
// ===== library: MasterCopy "Flow_Sensor" =====

FUNCTION_BLOCK "Flow_Sensor"   // FB1, FBD
TITLE = Pulsed Output Flow Accumlation
{ S7_Optimized_Access := 'TRUE' }
VERSION : 0.1
// Description: This function is used to Accumlate the flow passing through a pulsed-output flow sensor connected to the digital input channel with the address#Flow_Meter.
// Author: Ahmed Abd Alrahiem
// Email: a.abdalrahiem@gmail.com
// Last Modification Date: July 21, 2021
   VAR_INPUT
      Flow_Meter : Bool;   // The adress of the digital input channel which the Flow sensor is connected to
      pulses_per_litre : UInt;   // The number of pulses which the sesnor will provide after having one letre through it
      Reset : Bool;   // If set, the accumlated flow will be reset to 0
   END_VAR
   VAR_OUTPUT
      Accumlated_Flow : Real;   // The accumlated flow passing through the sensor
   END_VAR
   VAR RETAIN
      pos_edge1 : Bool;
      Flow_FB_counter_DB : CTU_UINT;
   END_VAR
   VAR_TEMP
      OF_DN : Bool;
      counted_pulses : UInt;
      Accumlated_Flow_temp : Real;
      Flow_base : Real;
      Flow_Delta : Real;
   END_VAR
   VAR_TEMP   // added for the SCL form of the ladder/FBD networks
      _w1 : Bool;
   END_VAR
BEGIN

REGION Network 1: Pulse Counting
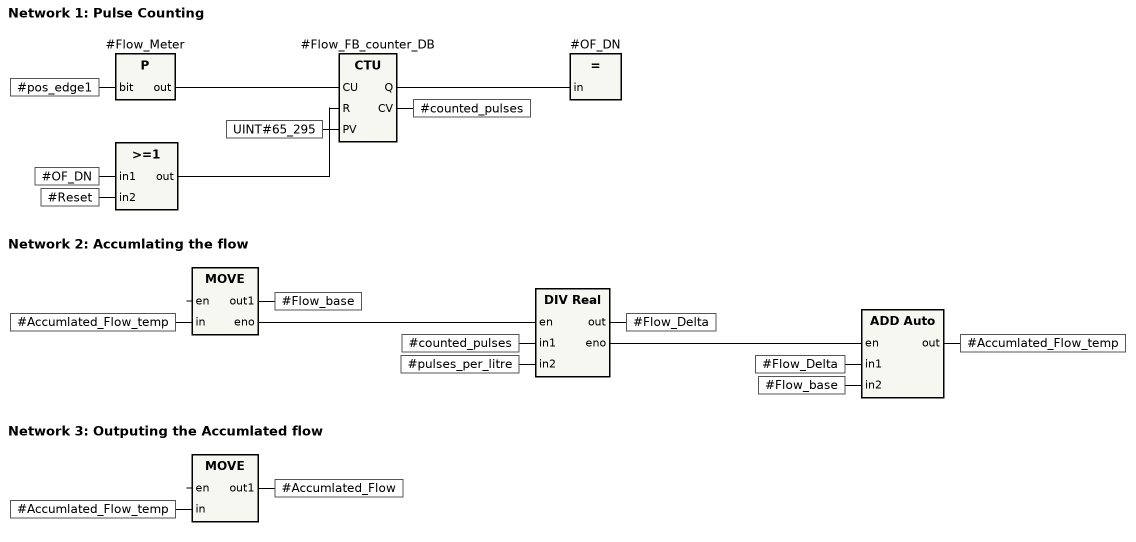
   #_w1 := #Flow_Meter AND NOT #pos_edge1;   // rising edge of #Flow_Meter
   #pos_edge1 := #Flow_Meter;
   #Flow_FB_counter_DB(CU := #_w1, R := #OF_DN OR #Reset, PV := UINT#65_295, CV => #counted_pulses);   // CTU
   #OF_DN := #Flow_FB_counter_DB.Q;
END_REGION

REGION Network 2: Accumlating the flow
   // The flow is accumlated, with integer overflow avoidance
   // ENO of a box is taken as its EN; it also drops when the box reports an error
   #Flow_base := #Accumlated_Flow_temp;
   #Flow_Delta := #counted_pulses / #pulses_per_litre;
   #Accumlated_Flow_temp := #Flow_Delta + #Flow_base;
END_REGION

REGION Network 3: Outputing the Accumlated flow
   #Accumlated_Flow := #Accumlated_Flow_temp;
END_REGION
END_FUNCTION_BLOCK

// ===== library: MasterCopy "Flow_Rate_Sensor" =====

FUNCTION_BLOCK "Flow_Rate_Sensor"   // FB2, FBD
TITLE = Flow rate calculation of a pulsed-output flow sensor
{ S7_Optimized_Access := 'TRUE' }
VERSION : 0.1
// Description: This function is used to calculate the frequecy of the pulses and convert it to the flow rate.
// Author: Ahmed Abd Alrahiem
// Email: a.abdalrahiem@gmail.com
// Last Modification Date: July 21, 2021
   VAR_INPUT
      Flow_Meter : Bool;   // The adress of the digital input channel which the Flow sensor is connected to
      "HZ_per_litre/min" : UInt;   // The proportionality constant between the pulse frequency and the flow rate
      Integration_Time : Time;   // The time window (in sec) used for flow rate calculation, it should be at least higher than the least possible pulse duration
   END_VAR
   VAR_OUTPUT
      Flow_Rate : Real;   // The flow rate of the stream passing through the sensor, calculated over the integration time
   END_VAR
   VAR RETAIN
      pos_edge1 : Bool;
      OF_DN : Bool;
      Flow_FB_counter_DB : CTU_UDINT;
      Flow_Rate_FB_Timer_DB : TP_TIME;
      Always_True : Bool := True;
   END_VAR
   VAR_TEMP
      Int_Time_DN : Bool;
      Integration_Time_Uint : UInt;
      Frequency : Real;
      counted_pulses : UDInt;
      counted_pulses_real : Real;
   END_VAR
   VAR_TEMP   // added for the SCL form of the ladder/FBD networks
      _w1 : Bool;
   END_VAR
BEGIN

REGION Network 1: Pulses counting
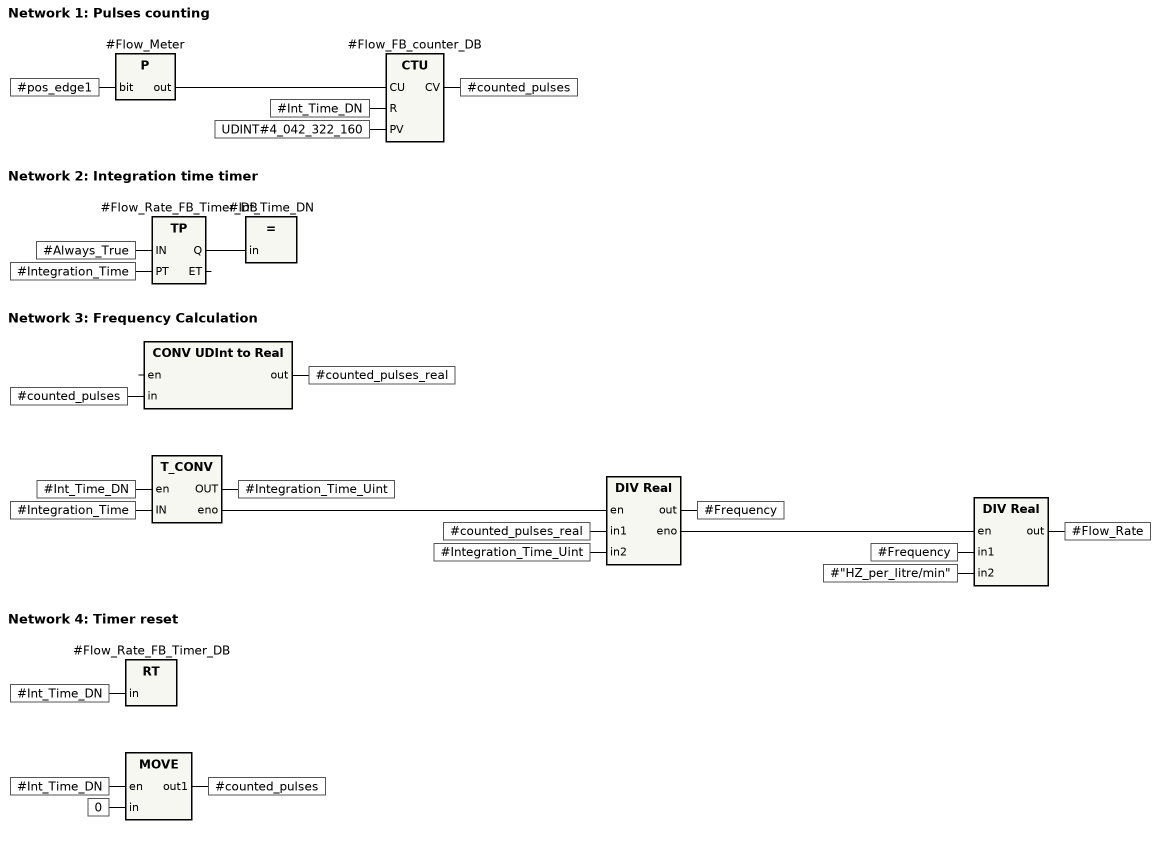
   #_w1 := #Flow_Meter AND NOT #pos_edge1;   // rising edge of #Flow_Meter
   #pos_edge1 := #Flow_Meter;
   #Flow_FB_counter_DB(CU := #_w1, R := #Int_Time_DN, PV := UDINT#4_042_322_160, CV => #counted_pulses);   // CTU
END_REGION

REGION Network 2: Integration time timer
   #Flow_Rate_FB_Timer_DB(IN := #Always_True, PT := #Integration_Time);   // TP
   #Int_Time_DN := #Flow_Rate_FB_Timer_DB.Q;
END_REGION

REGION Network 3: Frequency Calculation
   // ENO of a box is taken as its EN; it also drops when the box reports an error
   #counted_pulses_real := UDINT_TO_REAL(#counted_pulses);
   IF #Int_Time_DN THEN
       #Integration_Time_Uint := T_CONV(IN := #Integration_Time);
       #Frequency := #counted_pulses_real / #Integration_Time_Uint;
       #Flow_Rate := #Frequency / #"HZ_per_litre/min";
   END_IF;
END_REGION

REGION Network 4: Timer reset
   IF #Int_Time_DN THEN
       RESET_TIMER(#Flow_Rate_FB_Timer_DB);
       #counted_pulses := 0;
   END_IF;
END_REGION
END_FUNCTION_BLOCK